{attribute 'GeneratedUsingTerminal: KL6581-0002'}
{attribute addProperty BoxType "KL6581-0002"}
{attribute addProperty Id "Channel_1AT %Q*Channel_F7FDEFA00"}
{attribute addProperty CRC "858121603"}
{attribute addProperty Size "0"}
TYPE KL_3325E583 :
STRUCT
	{attribute addProperty Name "Channel_1"}
	Channel_1 : Channel_F7FDEFA0;
END_STRUCT
END_TYPE

(* stored: Version 1.2.0.0, ProductVersion 3.1.4024.9
   DUT KL_3325E583: Id {d205f0d2-6f7a-458d-8af2-7970a2615bb8} *)
